(* PLC project Stairs Light Control Example, CONTROLLINO GmbH CONTROLLINO MAXI Automation 0.1.0, author Firmware Team *)
(* stored: creationDateTime 2022-06-29T09:04:32, contentDescription Stairs light control example for CONTROLLINO MAXI Automation Outputs: DO0 -> %QX0.0 -> LIGHT_DOWN DO1 -> %QX0.1 -> LIGHT_MIDDLE DO2 -> %QX0.2 -> LIGHT_UP Inputs: AI2 -> %IX0.0 -> SWITCH_DOWN AI3 -> %IX0.1 -> SWITCH_UP AI4 -> %IX0.2 -> PRESENCE_SENSOR Behavior: The switches at both ends of the stairs are push buttons and will turn the lights on and off. The lights will turn on and off in sequence with a delay of N milliseconds. The lights will turn off after N seconds if no presence is detected on a sensor that is placed in the middle of the stairs. MIT License Copyright (c) 2016-2022 CONTROLLINO GmbH Permission is hereby granted, free of charge, to any person obtaining a copy of this software and associated documentation files (the "Software"), to deal in the Software without restriction, including without limitation the rights to use, copy, modify, merge, publish, distribute, sublicense, and/or sell copies of the Software, and to permit persons to whom the Software is furnished to do so, subject to the following conditions: The above copyright notice and this permission notice shall be included in all copies or substantial portions of the Software. THE SOFTWARE IS PROVIDED "AS IS", WITHOUT WARRANTY OF ANY KIND, EXPRESS OR IMPLIED, INCLUDING BUT NOT LIMITED TO THE WARRANTIES OF MERCHANTABILITY, FITNESS FOR A PARTICULAR PURPOSE AND NONINFRINGEMENT. IN NO EVENT SHALL THE AUTHORS OR COPYRIGHT HOLDERS BE LIABLE FOR ANY CLAIM, DAMAGES OR OTHER LIABILITY, WHETHER IN AN ACTION OF CONTRACT, TORT OR OTHERWISE, ARISING FROM, OUT OF OR IN CONNECTION WITH THE SOFTWARE OR THE USE OR OTHER DEALINGS IN THE SOFTWARE. CONTROLLINO - First software open-source PLC (ARDUINO compatible) https://controllino.com/ https://github.com/CONTROLLINO-PLC https://www.arduino.cc/ author: CONTROLLINO firmware team version: 0.1.0, modificationDateTime 2022-07-12T16:46:46, version 0.1.0 *)

PROGRAM inputs
  VAR
    AI2 AT %IX0.0 : BOOL;
    AI3 AT %IX0.1 : BOOL;
    AI4 AT %IX0.2 : BOOL;
  END_VAR
  VAR_EXTERNAL
    SWITCH_DOWN : BOOL;
    SWITCH_UP : BOOL;
    PRESENCE_SENSOR : BOOL;
  END_VAR

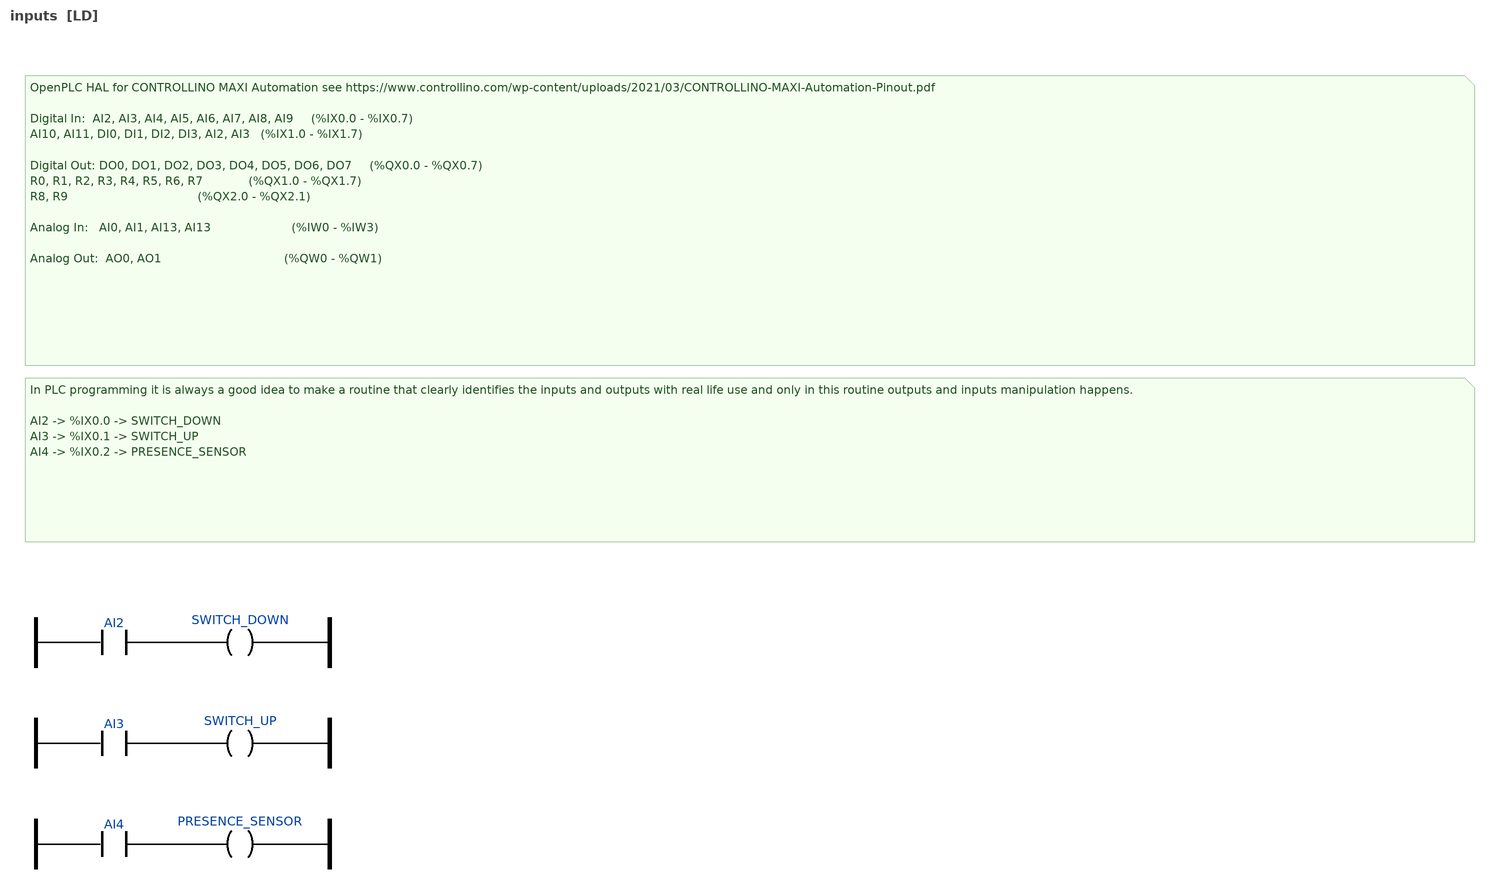
(* LD diagram, written out as Structured Text *)
(* OpenPLC HAL for CONTROLLINO MAXI Automation see https://www.controllino.com/wp-content/uploads/2021/03/CONTROLLINO-MAXI-Automation-Pinout.pdf

Digital In:  AI2, AI3, AI4, AI5, AI6, AI7, AI8, AI9     (%IX0.0 - %IX0.7)
             AI10, AI11, DI0, DI1, DI2, DI3, AI2, AI3   (%IX1.0 - %IX1.7)

Digital Out: DO0, DO1, DO2, DO3, DO4, DO5, DO6, DO7     (%QX0.0 - %QX0.7)
             R0, R1, R2, R3, R4, R5, R6, R7             (%QX1.0 - %QX1.7)
             R8, R9                                     (%QX2.0 - %QX2.1)

Analog In:   AI0, AI1, AI13, AI13                       (%IW0 - %IW3)

Analog Out:  AO0, AO1                                   (%QW0 - %QW1) *)
(* In PLC programming it is always a good idea to make a routine that clearly identifies the inputs and outputs with real life use and only in this routine outputs and inputs manipulation happens.

AI2 -> %IX0.0 -> SWITCH_DOWN
AI3 -> %IX0.1 -> SWITCH_UP
AI4 -> %IX0.2 -> PRESENCE_SENSOR *)
SWITCH_DOWN := AI2;
SWITCH_UP := AI3;
PRESENCE_SENSOR := AI4;
END_PROGRAM

PROGRAM control
  VAR_EXTERNAL
    SWITCH_DOWN : BOOL;
    SWITCH_UP : BOOL;
    PRESENCE_SENSOR : BOOL;
    LIGHT_DOWN : BOOL;
    LIGHT_MIDDLE : BOOL;
    LIGHT_UP : BOOL;
  END_VAR
  VAR
    T_SEQUENCE : TIME := T#500ms;
    T_OFF_LIGHTS : TIME := T#10s;
    LIGHT_CONTROL : BOOL;
    ENABLE_OFF_SWITCH : BOOL;
    DOWN_SEQUENCE : BOOL;
    UP_SEQUENCE : BOOL;
    TON1 : TON;
    TON2 : TON;
    TON3 : TON;
    TON4 : TON;
    TON0 : TON;
    TON5 : TON;
    TON6 : TON;
    TON7 : TON;
    TON8 : TON;
  END_VAR
  VAR  (* added by the conversion: wires and edge detectors of the diagram *)
    R_TRIG1 : R_TRIG;
    R_TRIG2 : R_TRIG;
    F_TRIG3 : F_TRIG;
    F_TRIG4 : F_TRIG;
    R_TRIG5 : R_TRIG;
    R_TRIG6 : R_TRIG;
    F_TRIG7 : F_TRIG;
    R_TRIG8 : R_TRIG;
    F_TRIG9 : F_TRIG;
    R_TRIG10 : R_TRIG;
    F_TRIG11 : F_TRIG;
    R_TRIG12 : R_TRIG;
    R_TRIG13 : R_TRIG;
    R_TRIG14 : R_TRIG;
    F_TRIG15 : F_TRIG;
    R_TRIG16 : R_TRIG;
    F_TRIG17 : F_TRIG;
  END_VAR

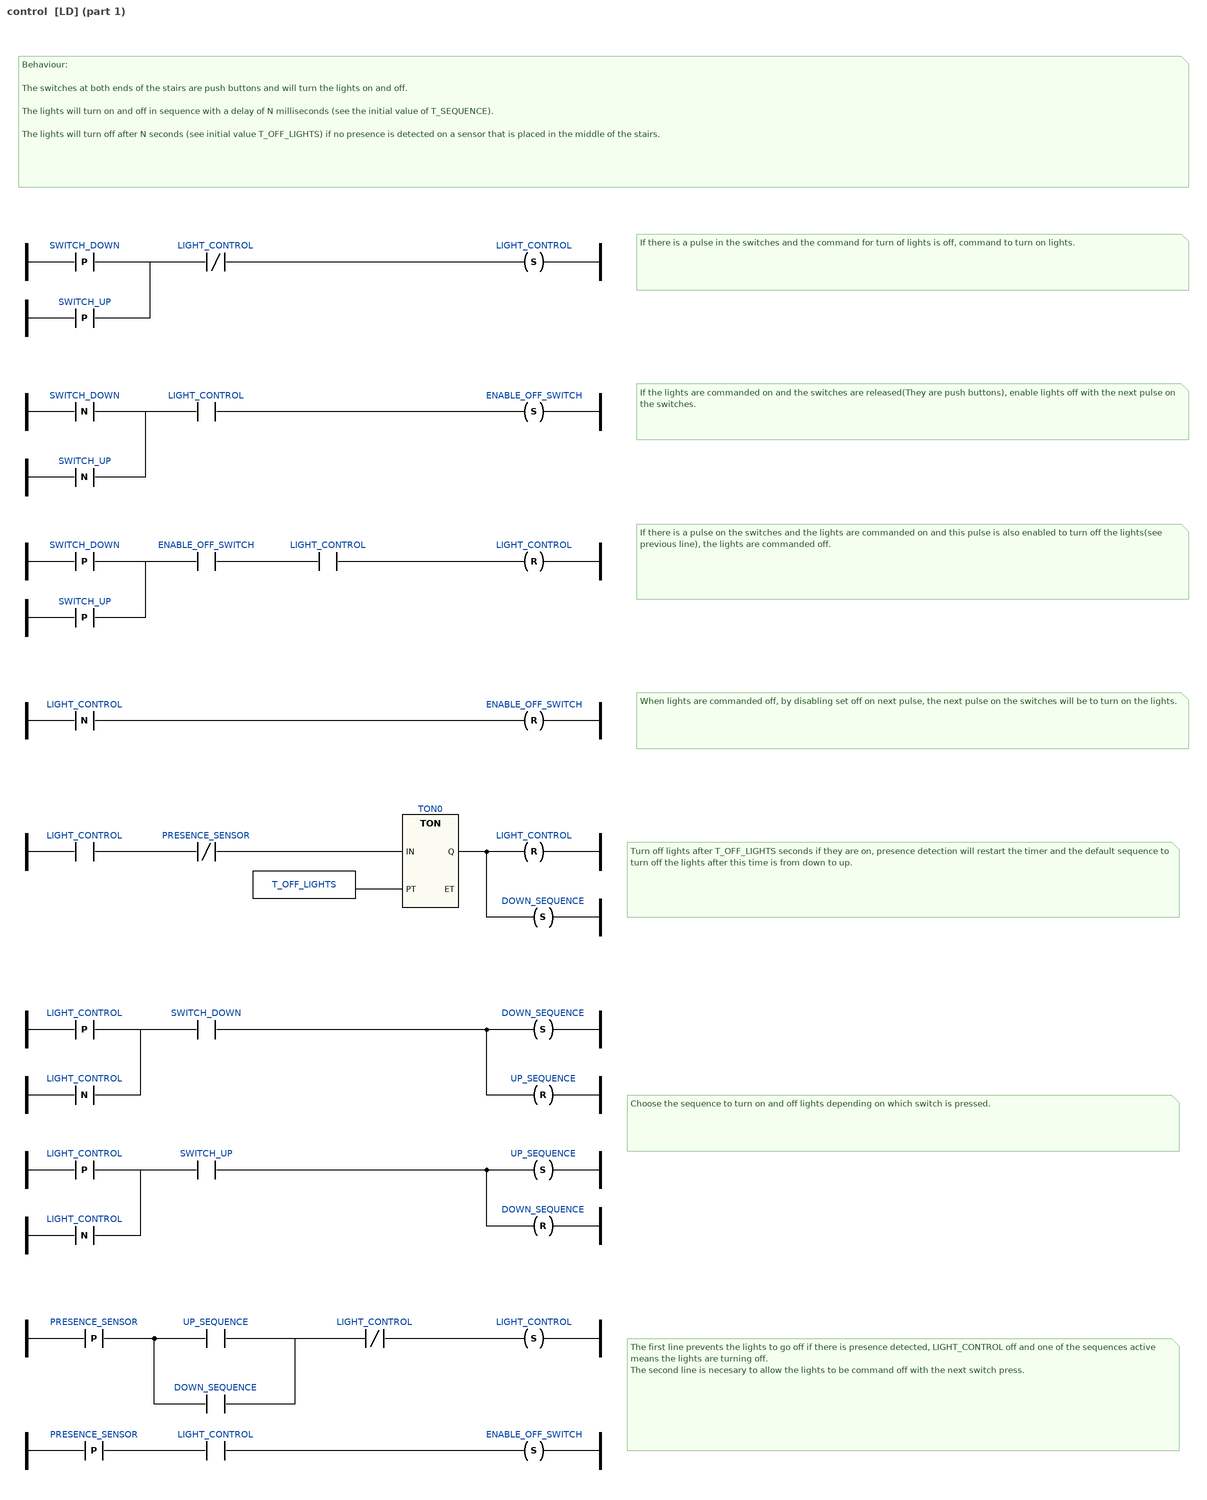
(* LD diagram, written out as Structured Text *)
(* Behaviour:

The switches at both ends of the stairs are push buttons and will turn the lights on and off.

The lights will turn on and off in sequence with a delay of N milliseconds (see the initial value of T_SEQUENCE).

The lights will turn off after N seconds (see initial value T_OFF_LIGHTS) if no presence is detected on a sensor that is placed in the middle of the stairs. *)
(* If there is a pulse in the switches and the command for turn of lights is off, command to turn on lights. *)
R_TRIG1(CLK := SWITCH_UP);
R_TRIG2(CLK := SWITCH_DOWN);
IF (R_TRIG1.Q OR R_TRIG2.Q) AND NOT LIGHT_CONTROL THEN LIGHT_CONTROL := TRUE; END_IF;
(* If the lights are commanded on and the switches are released(They are push buttons), enable lights off with the next pulse on the switches. *)
F_TRIG3(CLK := SWITCH_DOWN);
F_TRIG4(CLK := SWITCH_UP);
IF (F_TRIG3.Q OR F_TRIG4.Q) AND LIGHT_CONTROL THEN ENABLE_OFF_SWITCH := TRUE; END_IF;
(* If there is a pulse on the switches and the lights are commanded on and this pulse is also enabled to turn off the lights(see previous line), the lights are commanded off. *)
R_TRIG5(CLK := SWITCH_DOWN);
R_TRIG6(CLK := SWITCH_UP);
IF (R_TRIG5.Q OR R_TRIG6.Q) AND ENABLE_OFF_SWITCH AND LIGHT_CONTROL THEN LIGHT_CONTROL := FALSE; END_IF;
(* When lights are commanded off, by disabling set off on next pulse, the next pulse on the switches will be to turn on the lights. *)
F_TRIG7(CLK := LIGHT_CONTROL);
IF F_TRIG7.Q THEN ENABLE_OFF_SWITCH := FALSE; END_IF;
(* Turn off lights after T_OFF_LIGHTS seconds if they are on, presence detection will restart the timer and the default sequence to turn off the lights after this time is from down to up. *)
TON0(IN := LIGHT_CONTROL AND NOT PRESENCE_SENSOR, PT := T_OFF_LIGHTS);
IF TON0.Q THEN LIGHT_CONTROL := FALSE; END_IF;
IF TON0.Q THEN DOWN_SEQUENCE := TRUE; END_IF;
R_TRIG8(CLK := LIGHT_CONTROL);
F_TRIG9(CLK := LIGHT_CONTROL);
IF (R_TRIG8.Q OR F_TRIG9.Q) AND SWITCH_DOWN THEN DOWN_SEQUENCE := TRUE; END_IF;
IF (R_TRIG8.Q OR F_TRIG9.Q) AND SWITCH_DOWN THEN UP_SEQUENCE := FALSE; END_IF;
(* Choose the sequence to turn on and off lights depending on which switch is pressed. *)
R_TRIG10(CLK := LIGHT_CONTROL);
F_TRIG11(CLK := LIGHT_CONTROL);
IF (R_TRIG10.Q OR F_TRIG11.Q) AND SWITCH_UP THEN UP_SEQUENCE := TRUE; END_IF;
IF (R_TRIG10.Q OR F_TRIG11.Q) AND SWITCH_UP THEN DOWN_SEQUENCE := FALSE; END_IF;
R_TRIG12(CLK := PRESENCE_SENSOR);
IF R_TRIG12.Q AND (DOWN_SEQUENCE OR UP_SEQUENCE) AND NOT LIGHT_CONTROL THEN LIGHT_CONTROL := TRUE; END_IF;
(* The first line prevents the lights to go off if there is presence detected, LIGHT_CONTROL off and one of the sequences active means the lights are turning off.
The second line is necesary to allow the lights to be command off with the next switch press. *)
R_TRIG13(CLK := PRESENCE_SENSOR);
IF R_TRIG13.Q AND LIGHT_CONTROL THEN ENABLE_OFF_SWITCH := TRUE; END_IF;
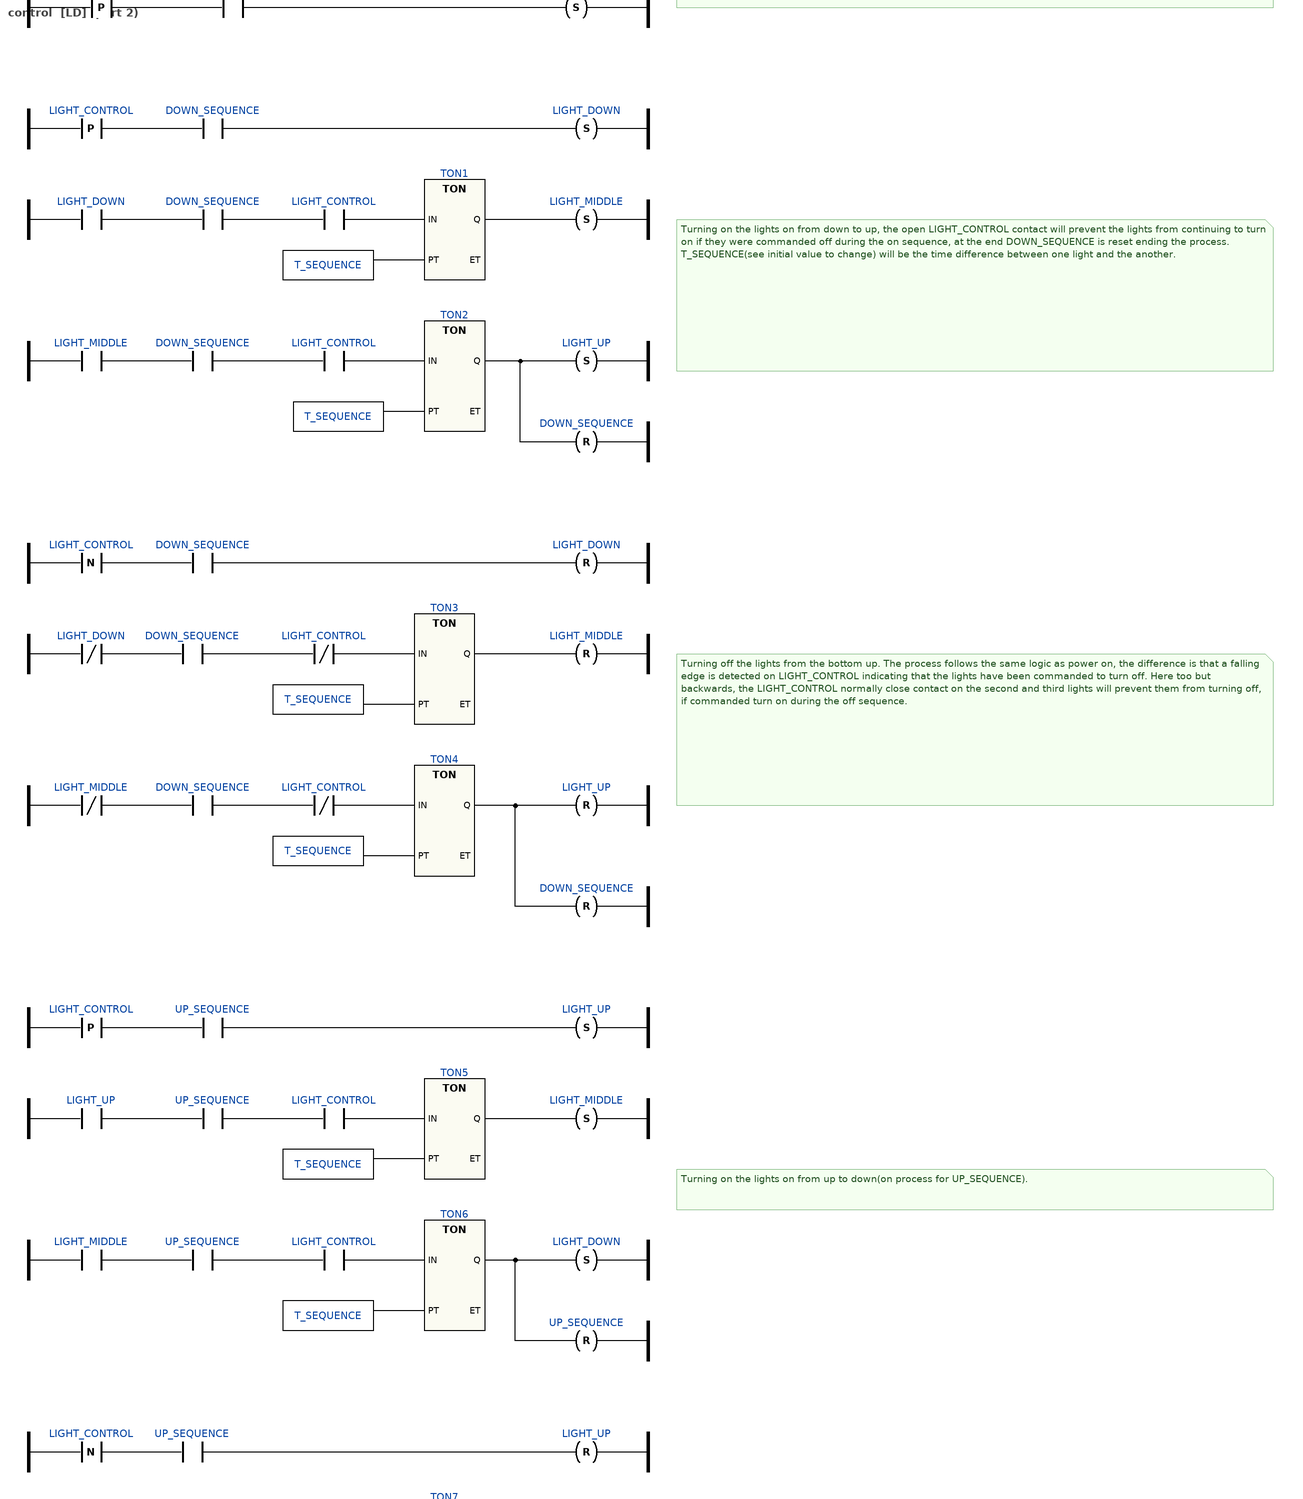
R_TRIG14(CLK := LIGHT_CONTROL);
IF R_TRIG14.Q AND DOWN_SEQUENCE THEN LIGHT_DOWN := TRUE; END_IF;
TON1(IN := LIGHT_DOWN AND DOWN_SEQUENCE AND LIGHT_CONTROL, PT := T_SEQUENCE);
IF TON1.Q THEN LIGHT_MIDDLE := TRUE; END_IF;
(* Turning on the lights on from down to up, the open LIGHT_CONTROL contact will prevent the lights from continuing to turn on if they were commanded off during the on sequence, at the end DOWN_SEQUENCE is reset ending the process.
T_SEQUENCE(see initial value to change) will be the time difference between one light and the another. *)
TON2(IN := LIGHT_MIDDLE AND DOWN_SEQUENCE AND LIGHT_CONTROL, PT := T_SEQUENCE);
IF TON2.Q THEN LIGHT_UP := TRUE; END_IF;
IF TON2.Q THEN DOWN_SEQUENCE := FALSE; END_IF;
F_TRIG15(CLK := LIGHT_CONTROL);
IF F_TRIG15.Q AND DOWN_SEQUENCE THEN LIGHT_DOWN := FALSE; END_IF;
TON3(IN := NOT LIGHT_DOWN AND DOWN_SEQUENCE AND NOT LIGHT_CONTROL, PT := T_SEQUENCE);
IF TON3.Q THEN LIGHT_MIDDLE := FALSE; END_IF;
(* Turning off the lights from the bottom up. The process follows the same logic as power on, the difference is that a falling edge is detected on LIGHT_CONTROL indicating that the lights have been commanded to turn off. Here too but backwards, the LIGHT_CONTROL normally close contact on the second and third lights will prevent them from turning off, if commanded turn on during the off sequence. *)
TON4(IN := NOT LIGHT_MIDDLE AND DOWN_SEQUENCE AND NOT LIGHT_CONTROL, PT := T_SEQUENCE);
IF TON4.Q THEN LIGHT_UP := FALSE; END_IF;
IF TON4.Q THEN DOWN_SEQUENCE := FALSE; END_IF;
R_TRIG16(CLK := LIGHT_CONTROL);
IF R_TRIG16.Q AND UP_SEQUENCE THEN LIGHT_UP := TRUE; END_IF;
TON5(IN := LIGHT_UP AND UP_SEQUENCE AND LIGHT_CONTROL, PT := T_SEQUENCE);
IF TON5.Q THEN LIGHT_MIDDLE := TRUE; END_IF;
(* Turning on the lights on from up to down(on process for UP_SEQUENCE). *)
TON6(IN := LIGHT_MIDDLE AND UP_SEQUENCE AND LIGHT_CONTROL, PT := T_SEQUENCE);
IF TON6.Q THEN LIGHT_DOWN := TRUE; END_IF;
IF TON6.Q THEN UP_SEQUENCE := FALSE; END_IF;
F_TRIG17(CLK := LIGHT_CONTROL);
IF F_TRIG17.Q AND UP_SEQUENCE THEN LIGHT_UP := FALSE; END_IF;
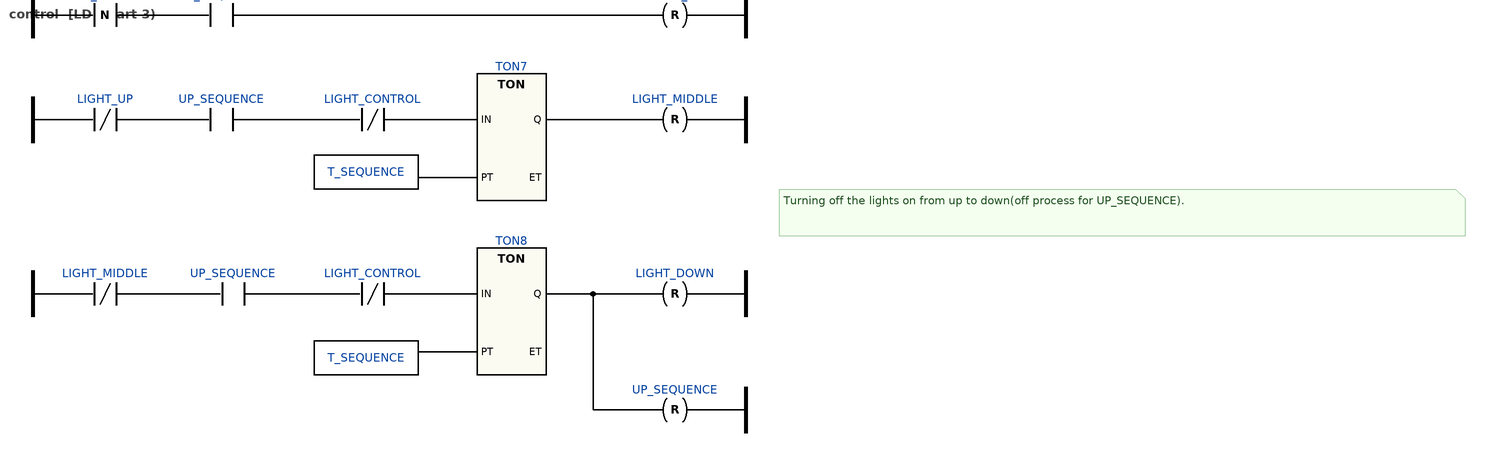
TON7(IN := NOT LIGHT_UP AND UP_SEQUENCE AND NOT LIGHT_CONTROL, PT := T_SEQUENCE);
IF TON7.Q THEN LIGHT_MIDDLE := FALSE; END_IF;
(* Turning off the lights on from up to down(off process for UP_SEQUENCE). *)
TON8(IN := NOT LIGHT_MIDDLE AND UP_SEQUENCE AND NOT LIGHT_CONTROL, PT := T_SEQUENCE);
IF TON8.Q THEN LIGHT_DOWN := FALSE; END_IF;
IF TON8.Q THEN UP_SEQUENCE := FALSE; END_IF;
END_PROGRAM

PROGRAM outputs
  VAR
    DO0 AT %QX0.0 : BOOL;
    DO1 AT %QX0.1 : BOOL;
    DO2 AT %QX0.2 : BOOL;
  END_VAR
  VAR_EXTERNAL
    LIGHT_DOWN : BOOL;
    LIGHT_MIDDLE : BOOL;
    LIGHT_UP : BOOL;
  END_VAR

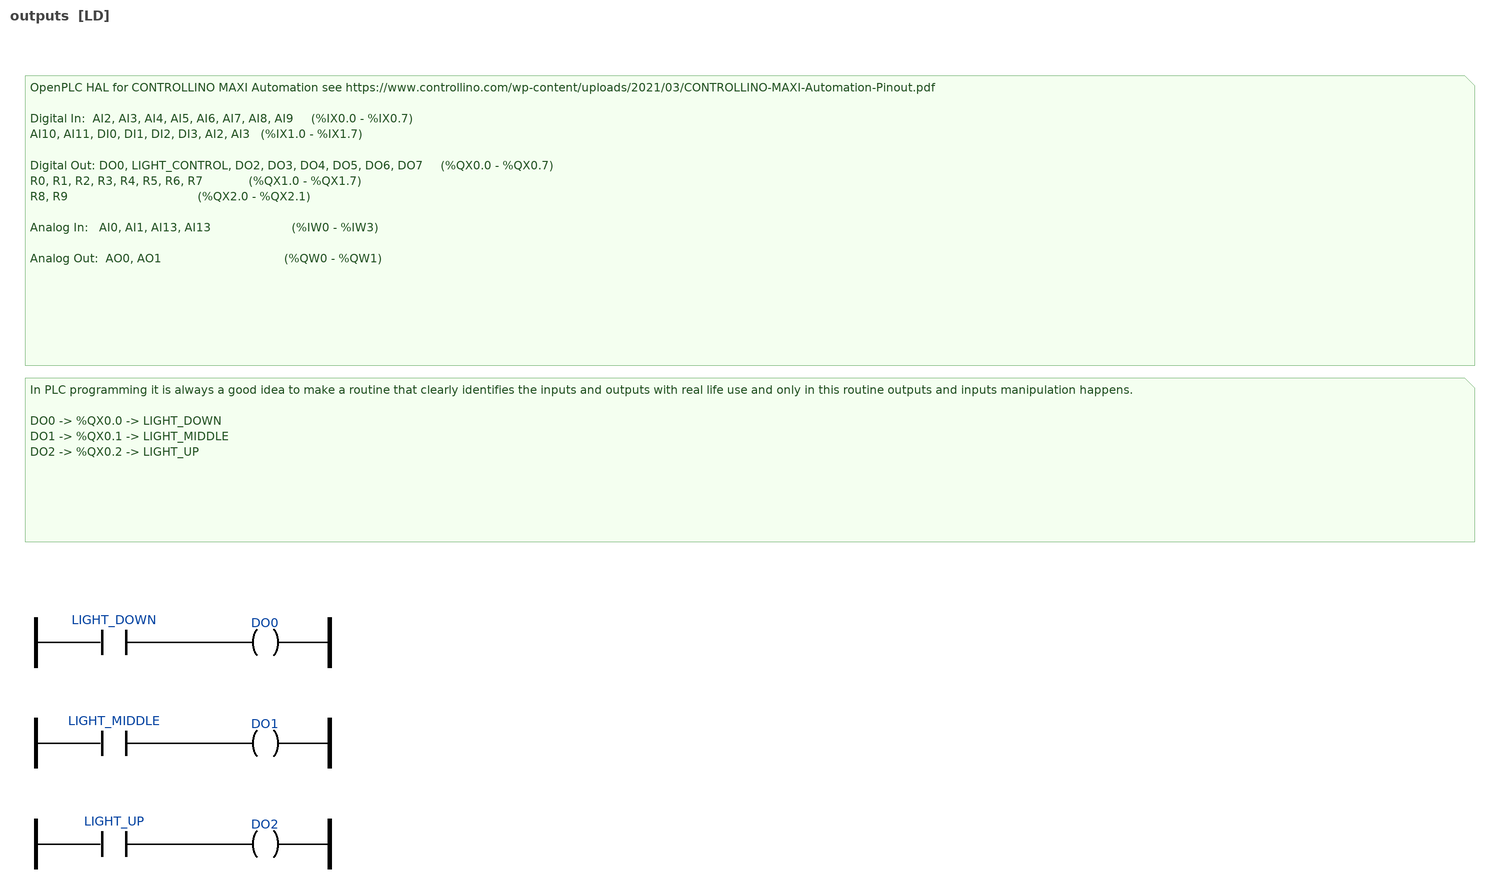
(* LD diagram, written out as Structured Text *)
(* OpenPLC HAL for CONTROLLINO MAXI Automation see https://www.controllino.com/wp-content/uploads/2021/03/CONTROLLINO-MAXI-Automation-Pinout.pdf

Digital In:  AI2, AI3, AI4, AI5, AI6, AI7, AI8, AI9     (%IX0.0 - %IX0.7)
             AI10, AI11, DI0, DI1, DI2, DI3, AI2, AI3   (%IX1.0 - %IX1.7)

Digital Out: DO0, LIGHT_CONTROL, DO2, DO3, DO4, DO5, DO6, DO7     (%QX0.0 - %QX0.7)
             R0, R1, R2, R3, R4, R5, R6, R7             (%QX1.0 - %QX1.7)
             R8, R9                                     (%QX2.0 - %QX2.1)

Analog In:   AI0, AI1, AI13, AI13                       (%IW0 - %IW3)

Analog Out:  AO0, AO1                                   (%QW0 - %QW1) *)
(* In PLC programming it is always a good idea to make a routine that clearly identifies the inputs and outputs with real life use and only in this routine outputs and inputs manipulation happens.

DO0 -> %QX0.0 -> LIGHT_DOWN
DO1 -> %QX0.1 -> LIGHT_MIDDLE
DO2 -> %QX0.2 -> LIGHT_UP *)
DO0 := LIGHT_DOWN;
DO1 := LIGHT_MIDDLE;
DO2 := LIGHT_UP;
END_PROGRAM

CONFIGURATION Config0
  RESOURCE Res0 ON PLC
    VAR_GLOBAL
      SWITCH_DOWN : BOOL;
      SWITCH_UP : BOOL;
      PRESENCE_SENSOR : BOOL;
      LIGHT_DOWN : BOOL;
      LIGHT_MIDDLE : BOOL;
      LIGHT_UP : BOOL;
    END_VAR
    TASK task0(INTERVAL := T#20ms, PRIORITY := 0);
    PROGRAM instance0 WITH task0 : inputs;
    PROGRAM instance1 WITH task0 : control;
    PROGRAM instance2 WITH task0 : outputs;
  END_RESOURCE
END_CONFIGURATION
